PROGRAM P_ModeSelector
VAR
	
END_VAR

//***********************************************************************************
//
// ETH Zürich / Robotic Fabrication Lab
// HIB C 13 / Stefano-Franscini-Platz 1
// CH-8093 Zürich
// 
// ***********************************************************************************
// 
// PROJECT     :  A061 Digital Casting System
// 
// FUNCTION    :  selector for mode control
// 
// AUTHOR      :  Weiting Chen
// 
// EMAIL       :  
// 
// Copyright   : 
//
// ***********************************************************************************


GVL_VAR.b_Mode_Manual := GVL_IO.ib_CC1_Button_Mode_Manual;
GVL_VAR.b_Mode_Laptop := GVL_IO.ib_CC1_Button_Mode_Laptop;

END_PROGRAM

(* stored: Version 1.1.0.1, ProductVersion 3.1.4024.11
   POU P_ModeSelector: Id {0eb7d8c2-292e-4a26-bb54-34c9ce7294b6}, SpecialFunc None *)
